FUNCTION_BLOCK FB_ModbusSlave IMPLEMENTS I_ModbusSlave
VAR
	iUnitID	:	BYTE; // address of the Slave
	arrAddressRead	:	ARRAY [0..50] OF ARRAY [0..2] OF WORD;
	(*arrAddressRead[x][y]: +x : index of Region Read.  arrAddressRead[0]: the first region Read.
							+y:
								case y of
									0: Register address for Read
									1: Number of register for read
									2: Function Read
					 *)
	iNumAddRegionRead	:	UINT;
	
	arrAddressWrite		: ARRAY [0..20] OF ARRAY [0..10] OF WORD;// write Multiple or single register
	(* the 20 is max number of region write,
		arrAddressWrite[x][y] : +x: index of Region Read.  arrAddressRead[0]: the first region Read. 
								+y:
									case y of
										0 :  Register address for Write
										1 : number of register will be write => modbus master automatic choose Function Write( single Register or Multi Regiseter)
										2..9 : max 8 value for write
										10: Write Function : e.g E_ModbusFunction.WriteSingleCoil
															
	*)
	iNumAddRegionWrite	: UINT;
	sName				:		STRING;
	bFirstCycle 		: 		BOOL := TRUE;
	iModbusErrorID		:		MODBUS_ERRORS;
END_VAR

PROPERTY AddressRead : POINTER TO WORD
GET
AddressRead := ADR(arrAddressRead);
END_GET
END_PROPERTY

PROPERTY AddressWrite : POINTER TO WORD
GET
AddressWrite := ADR( arrAddressWrite);
END_GET
END_PROPERTY

METHOD Convert : BOOL
VAR_INPUT
	iRegionNo	:	INT;
	pReadData	:	POINTER TO word;
END_VAR
END_METHOD

METHOD FirstCycle // must be call once time 
VAR_INPUT
	sName : STRING;
	iUnitID : BYTE ; // modbus address of the device : 1- 255
END_VAR
THIS^.sName := sName;
THIS^.iUnitID := iUnitID;
END_METHOD

{attribute 'monitoring' := 'variable'}
PROPERTY ModbusErrorID : MODBUS_ERRORS
GET
ModbusErrorID := iModbusErrorID;
END_GET
SET
iModbusErrorID := ModbusErrorID;
END_SET
END_PROPERTY

PROPERTY Name : STRING
GET
Name := sName;
END_GET
SET
sName := Name;
END_SET
END_PROPERTY

PROPERTY NumAddRegionRead : UINT
GET
NumAddRegionRead := iNumAddRegionRead;
END_GET
END_PROPERTY

PROPERTY NumAddRegionWrite : UINT
GET
NumAddRegionWrite := iNumAddRegionWrite;
END_GET
END_PROPERTY

PROPERTY UnitID : BYTE
GET
UnitID := iUnitID;
END_GET
SET
iUnitID := UnitID;
END_SET
END_PROPERTY

END_FUNCTION_BLOCK

(* stored: Version 1.1.0.1, ProductVersion 3.1.4024.12
   POU FB_ModbusSlave: Id {3c28a97a-7b9e-4799-881a-cc6e3fde9dc8}, SpecialFunc None
   Property AddressRead: Id {6bad1251-2173-4dad-ba55-b0ca54c51b4b}
   Get Get: Id {985bce2e-167a-45be-8089-4bec8ed22891}
   Property AddressWrite: Id {5c4258fd-a88b-4ea9-9dad-ce3ab400d74c}
   Get Get: Id {a0e8c4bf-b72b-4849-87ca-51e8c4ef32ff}
   Method Convert: Id {3fd4f7ca-261b-4d44-a547-551bb3314b31}
   Method FirstCycle: Id {5bee89eb-ef51-45da-b0f8-e42cc2ee867a}
   Property ModbusErrorID: Id {10a0f1de-4a02-4f0a-b4da-6536bf3ef75c}
   Get Get: Id {feb78e1e-5a56-48eb-bc4b-7b331dd98e5f}
   Set Set: Id {41376bb8-baa5-43b9-b4af-8506bc2623c3}
   Property Name: Id {06664f22-c56c-4b15-a1d7-a34951a97f8f}
   Get Get: Id {9022ba2a-8142-4b11-aa2b-314496623ffe}
   Set Set: Id {6f38bf1f-ebc9-4220-aa3d-695fb0fa3d27}
   Property NumAddRegionRead: Id {b5abfa30-10e8-4954-8477-81f742d0936e}
   Get Get: Id {f25e2842-516b-4ae1-85e4-95db72ca8802}
   Property NumAddRegionWrite: Id {969a2335-93c3-4c90-91d6-c32d995f4ac2}
   Get Get: Id {b1adea90-2fa2-4e92-a2fc-89d69ec231dc}
   Property UnitID: Id {09876766-f5af-4b25-9fd2-4a972765efd0}
   Get Get: Id {cd055b1c-cf68-47e9-b9fd-fac9e0785529}
   Set Set: Id {0fe61a22-da1d-49e5-a05a-46b09e346e4b} *)
